FUNCTION_BLOCK CTRL_PID_AR (* AR-Adapter-Wrapper um OSCAT CTRL_PID - bruckt zwischen adapter und OSCAT PID-Regler. Istwert, Sollwert, Hand-Umschaltung, Handwert, Reglerparameter UND Rauschunterdrueckung/Offset/Grenzwerte vollstaendig als Adapter-Sockets - kein explizites REQ mehr noetig. *)
  (* Standard: 61499-2; Description: Copyright (c) 2026 Meisterschulen am Ostbahnhof This program and the accompanying materials are made available under the terms of the Eclipse Public License 2.0 which is available at https://www.eclipse.org/legal/epl-2.0/ SPDX-License-Identifier: EPL-2.0 *)
  (* Version 1.4, 2026-10-03, Franz Höpfinger, Meisterschulen am Ostbahnhof, Franz: 'die Eingaenge sollen identisch sortiert sein wie bei dem enthaltenen FB' - Sockets (inkl. EventConnections/DataConnections/Dokumentation) auf die Reihenfolge von CTRL_PID.InputVars umsortiert: AR_ACT, SET, SUP, OFS, M_I, AX_MAN, KP, TN, TV, LL, LH (vorher: AR_ACT, SET, AX_MAN, M_I, KP, TN, TV, SUP, OFS, LL, LH - SUP/OFS/LL/LH waren beim v1.3-Umbau einfach hinten angehaengt worden). Rein kosmetisch/strukturell, keine funktionale Aenderung. *)
  (* Version 1.3, 2026-10-03, Franz Höpfinger, Meisterschulen am Ostbahnhof, Franz: 'SUP, OFS, LL, LH muessen auch AR Adapter werden, wie KP und TN. REQ faellt dann weg, RST bleibt. CNF entfaellt auch.' - SUP/OFS/LL/LH von InputVars (REAL, With-gebunden an REQ) auf AR-Adapter-Sockets umgestellt (gleiches Muster wie KP/TN/TV/M_I: *.E1 loest CTRL_PID.REQ aus, *.D1 liefert den Wert). Explizites REQ-EventInput (inkl. With-Bindungen) und CNF-EventOutput komplett entfernt - CTRL_PID.CNF->E_D_FF_ANY.CLK bleibt intern bestehen (fuer das Latch von Y/DIFF/LIM), nur der externe CNF-Durchgriff entfaellt. RST unveraendert. *)
  (* Version 1.2, 2026-09-19, Franz Höpfinger, Meisterschulen am Ostbahnhof, Bugfix: REQ hatte keine With-Verknuepfung zu SUP/OFS/LL/LH (IEC 61499 - ungebundene Vars werden nicht zuverlaessig gelesen), jetzt ergaenzt, gespiegelt vom inneren CTRL_PID. M_I/KP/TN/TV von InputVars auf AR-Adapter-Sockets umgestellt (Konsistenz mit AR_ACT/SET). *)
  (* Version 1.1, 2026-09-12, Franz Höpfinger, Meisterschulen am Ostbahnhof, INIT/INITO entfernt (CTRL_PID kennt kein INIT, nur REQ/RST) - stattdessen echtes REQ-EventInput/CNF-EventOutput ergaenzt, direkt auf CTRL_PID.REQ/CNF gemappt. SET von InputVar auf AR-Socket umgestellt (dynamisch berechneter Sollwert, wie AR_ACT) - SET.E1 triggert CTRL_PID.REQ zusaetzlich zu AR_ACT.E1/AX_MAN.E1. *)
  (* Version 1.0, 2026-09-12, Franz Höpfinger, Meisterschulen am Ostbahnhof, Initial implementation of CTRL_PID_AR wrapper FB *)
  PACKAGE OSCAT_adapter::Control;
  (* Documentation:
  CTRL_PID_AR
   🇩🇪 Deutsch
   AR-Adapter-Wrapper um OSCAT::Basic::POUs::Engineering::Control::CTRL_PID. Istwert (AR_ACT), Sollwert (SET), Rauschunterdrueckung/Offset (SUP/OFS), Handwert (M_I), Handbetrieb-Umschaltung (AX_MAN), Reglerparameter (KP/TN/TV) UND Grenzwerte (LL/LH) sind als Adapter-Sockets ausgefuehrt, in derselben Reihenfolge wie die InputVars des umschlossenen CTRL_PID - jeder loest bei Ankunft eines neuen Werts CTRL_PID.REQ aus. Kein explizites REQ-Event mehr noetig, da jeder Socket selbst triggert. RST (Reset des Integrators) bleibt als eigenes Event erhalten.
   Reine Adapter-Grenze
    - AR_ACT (Socket, AR): Istwert (REAL, z. B. von FT_DERIV_10_AR.AR_OUT)
   - SET (Socket, AR): Sollwert (REAL, dynamisch berechnet, z. B. Fahrgeschwindigkeit*Voreilung)
   - SUP (Socket, AR): Rauschunterdrueckung (REAL, dynamisch)
   - OFS (Socket, AR): Offset (REAL, dynamisch)
   - M_I (Socket, AR): Handwert (REAL, dynamisch)
   - AX_MAN (Socket, AX): Handbetrieb-Umschaltung (optional, z. B. von AX_T_FF.Q)
   - KP/TN/TV (Socket, AR): Reglerparameter (REAL, dynamisch)
   - LL/LH (Socket, AR): unterer/oberer Grenzwert (REAL, dynamisch)
   - AR_Y (Plug, AR): Stellwert (REAL, z. B. zur Weitergabe an AR_TO_AD_NUM.AR_IN)
   - AR_DIFF (Plug, AR): Regelabweichung (DIFF = SET - ACT, REAL)
   - AB_LIM (Plug, AB): Begrenzung aktiv Flag (LIM, BOOL)
    🇬🇧 English
   AR-adapter wrapper around OSCAT::Basic::POUs::Engineering::Control::CTRL_PID. Actual value (AR_ACT), set point (SET), noise suppression/offset (SUP/OFS), manual value (M_I), manual mode switch (AX_MAN), controller gains (KP/TN/TV) AND limits (LL/LH) are all adapter sockets, in the same order as the wrapped CTRL_PID's own InputVars, each triggering CTRL_PID.REQ on arrival - no explicit REQ event needed any more, since every socket triggers itself. RST (integrator reset) remains its own event. Control output (AR_Y), control error (AR_DIFF) and limit flag (AB_LIM) are adapter plugs.
  *)
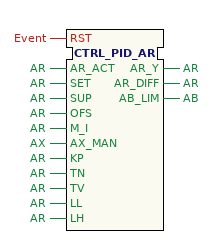
  EVENT_INPUT
    RST; (* Reset des Integrators (durchgereicht an CTRL_PID.RST) *)
  END_EVENT
  SOCKETS
    AR_ACT : adapter::types::unidirectional::AR; (* Istwert (REAL) *)
    SET : adapter::types::unidirectional::AR; (* Sollwert (REAL, dynamisch berechnet) *)
    SUP : adapter::types::unidirectional::AR; (* Rauschunterdrueckung (REAL, dynamisch) *)
    OFS : adapter::types::unidirectional::AR; (* Offset (REAL, dynamisch) *)
    M_I : adapter::types::unidirectional::AR; (* Handwert (REAL, dynamisch) *)
    AX_MAN : adapter::types::unidirectional::AX; (* Handbetrieb Umschaltung (BOOL/Event, optional) *)
    KP : adapter::types::unidirectional::AR; (* Proportionalbeiwert (REAL, dynamisch) *)
    TN : adapter::types::unidirectional::AR; (* Nachstellzeit (REAL, dynamisch) *)
    TV : adapter::types::unidirectional::AR; (* Vorhaltzeit (REAL, dynamisch) *)
    LL : adapter::types::unidirectional::AR; (* Unterer Grenzwert (REAL, dynamisch) *)
    LH : adapter::types::unidirectional::AR; (* Oberer Grenzwert (REAL, dynamisch) *)
  END_SOCKETS
  PLUGS
    AR_Y : adapter::types::unidirectional::AR; (* Stellwert (REAL) *)
    AR_DIFF : adapter::types::unidirectional::AR; (* Regelabweichung / Differenz (REAL) *)
    AB_LIM : adapter::types::unidirectional::AB; (* Begrenzung aktiv Flag (BOOL) *)
  END_PLUGS
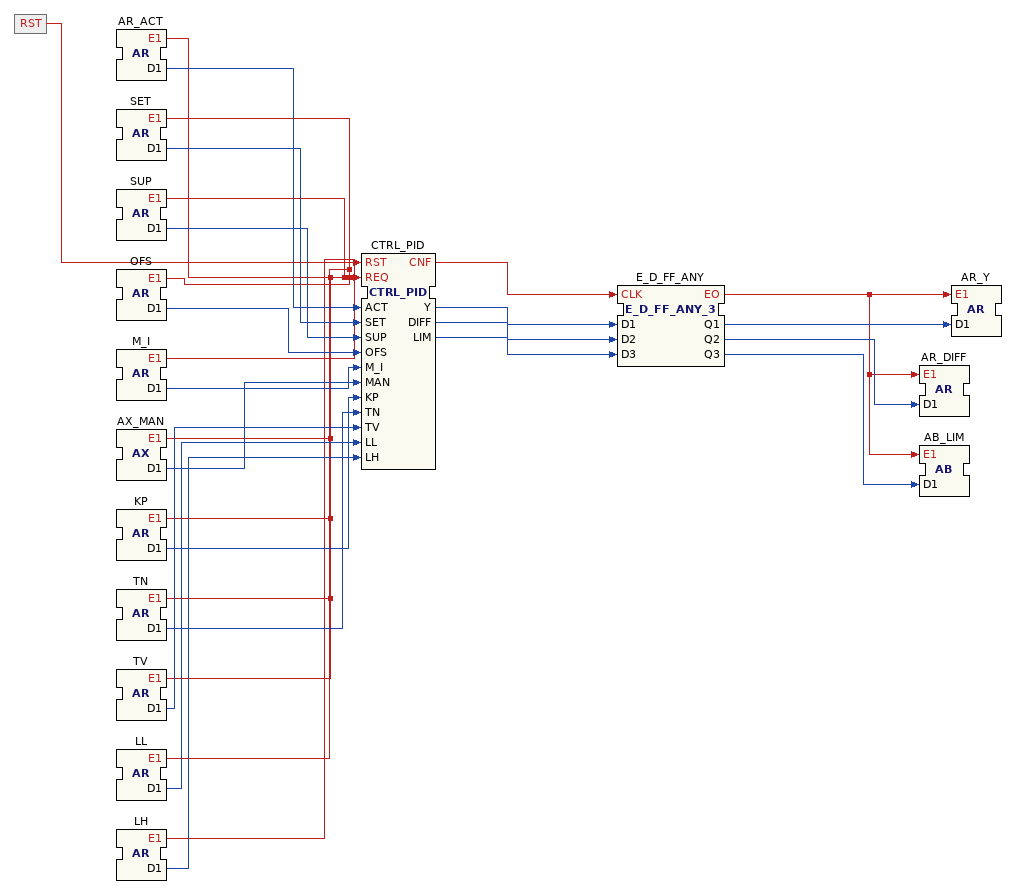
  FBS
    CTRL_PID : OSCAT::Basic::POUs::Engineering::Control::CTRL_PID;
    E_D_FF_ANY : iec61499::events::E_D_FF_ANY_3;
  END_FBS
  EVENT_CONNECTIONS
    RST TO CTRL_PID.RST;
    AR_ACT.E1 TO CTRL_PID.REQ;
    SET.E1 TO CTRL_PID.REQ;
    SUP.E1 TO CTRL_PID.REQ;
    OFS.E1 TO CTRL_PID.REQ;
    M_I.E1 TO CTRL_PID.REQ;
    AX_MAN.E1 TO CTRL_PID.REQ;
    KP.E1 TO CTRL_PID.REQ;
    TN.E1 TO CTRL_PID.REQ;
    TV.E1 TO CTRL_PID.REQ;
    LL.E1 TO CTRL_PID.REQ;
    LH.E1 TO CTRL_PID.REQ;
    CTRL_PID.CNF TO E_D_FF_ANY.CLK;
    E_D_FF_ANY.EO TO AR_Y.E1;
    E_D_FF_ANY.EO TO AR_DIFF.E1;
    E_D_FF_ANY.EO TO AB_LIM.E1;
  END_CONNECTIONS
  DATA_CONNECTIONS
    AR_ACT.D1 TO CTRL_PID.ACT;
    SET.D1 TO CTRL_PID.SET;
    SUP.D1 TO CTRL_PID.SUP;
    OFS.D1 TO CTRL_PID.OFS;
    M_I.D1 TO CTRL_PID.M_I;
    AX_MAN.D1 TO CTRL_PID.MAN;
    KP.D1 TO CTRL_PID.KP;
    TN.D1 TO CTRL_PID.TN;
    TV.D1 TO CTRL_PID.TV;
    LL.D1 TO CTRL_PID.LL;
    LH.D1 TO CTRL_PID.LH;
    CTRL_PID.Y TO E_D_FF_ANY.D1;
    CTRL_PID.DIFF TO E_D_FF_ANY.D2;
    CTRL_PID.LIM TO E_D_FF_ANY.D3;
    E_D_FF_ANY.Q1 TO AR_Y.D1;
    E_D_FF_ANY.Q2 TO AR_DIFF.D1;
    E_D_FF_ANY.Q3 TO AB_LIM.D1;
  END_CONNECTIONS
END_FUNCTION_BLOCK
